{attribute 'TcGenerated'}
{attribute 'no-analysis'}
{attribute 'linkalways'}
// This function has been automatically generated from the project information.
VAR_GLOBAL CONSTANT
	{attribute 'const_non_replaced'}
	stLibVersion_MqttFramework : ST_LibVersion := (iMajor := 1, iMinor := 0, iBuild := 0, iRevision := 0, nFlags := 0, sVersion := '1.0.0.0');
END_VAR

(* stored: Version 1.1.0.1, ProductVersion 3.1.4024.0
   GVL Global_Version: Id {44caf57d-6026-4248-80ad-efd771b04111} *)
